///////////
// Structure For Jema Module 
//////////
TYPE PowerCol :
STRUCT
		MesP 						: REAL; 		// {1}(kW) Active Power output (AC) of PCS
		MesQ 						: REAL; 		// {1}(kVAr) Reactive AC Power Produced by PCS 
		MesPdc						: REAL ; 		// {1}(kW) DC Power . 
		MesCosPhi 					: REAL;  		// {0}(p.u) Power factor
		MesFreq						: REAL ; 		// {0}(Hz) Frequency
		MesTemp						: REAL ; 		// {0}(°C) PCS Internal Temperature
		MesU 						: REAL;  		// {0}(V) AC Voltage measure
		MesUdc 						: REAL;  		// {0}(V) DC Voltage measure
		MesI 						: REAL; 		// {0}(A) Total AC current 
		MesI1						: REAL ; 		// {0}(A) Phase 1 AC Current
		MesI2						: REAL ;        // {0}(A) Phase 2 AC Current
		MesI3						: REAL ;        // {0}(A) Phase 3 AC Current
		MesIdc 						: REAL; 		// {0}(A) Total DC current from batteries (+ = discharge)
		MesPavailable 				: REAL;  		// {1}(kW) Available PCS Power 
		MesPconnected				: REAL ; 		// {0}(kW) Connected PCS Power 
		MesDcSwitchClosed			: BOOL ; 		// {0}(NA) Position of the DC Switch : True = Switch closed
		MesAcSwitchClosed			: BOOL ; 		// {0}(NA) Position of the AC Switch : True = Switch closed
		MesTempControl      		: REAL ; 		// {0}(°C) Temperature of control card
		MesTempPowerUnit    		: REAL ;		// {0}(°C) Temperature of Power Unit
		MesTempCabinet      		: REAL ; 		// {0}(°C) Cabinet temperature
		MesTempCoil1        		: REAL ; 		// {0}(°C) Coil temperature
		MesRegAlarm0        		: WORD ; 		// {0}Alarm Word of PCS
		MesRegAlarm1        		: WORD ; 		// {0}Alarm Word of PCS 
		MesRegAlarm2        		: WORD ; 		// {0}Alarm Word of PCS 
		MesRegAlarm3        		: WORD ;  		// {0}Alarm Word of PCS
		MesRegAlarm4        		: WORD ;  		// {0}Alarm Word of PCS
		MesDeratingWord				: WORD ;		// {0}Derating word of PCS
		MesHeartbit					: REAL ;		// {0}Heartbit
		MesDoorOpened				: BOOL ;		// {1}Door of the Power module is opened	
		
		MesJemaAlarms				: PowerCol_JemaAlarms;

			

END_STRUCT
END_TYPE

(* stored: Version 1.1.0.1, ProductVersion 3.1.4024.9
   DUT PowerCol: Id {8fc4c86f-db8d-4330-a05b-4057e06fe46c} *)
